// TwinCAT 3 PLC project pruebaFiltrado
// ProgramVersion: 3.1.4024.0
// libraries:
//   Tc2_Standard, * (Beckhoff Automation GmbH)
//   Tc2_System, * (Beckhoff Automation GmbH)
//   Tc3_Module, * (Beckhoff Automation GmbH)
// project tree:
//   GVLs/ GVLvars.TcGVL
//   / PlcTask.TcTTO
//   POUs/ MAIN.TcPOU
// real-time tasks:
//   TASK PlcTask: cycle T#10ms, priority 20, ADS port 350

CONFIGURATION pruebaFiltrado
    RESOURCE PLC ON TwinCAT3
        TASK PlcTask(INTERVAL := T#10ms, PRIORITY := 20);
        PROGRAM MAIN WITH PlcTask : MAIN;
    END_RESOURCE
END_CONFIGURATION

// ---- GVLs/GVLvars.TcGVL
{attribute 'qualified_only'}
VAR_GLOBAL
	// Cuadro
	{attribute 'OPC.UA.DA' := '1'}
	botonStart : BOOL;
	
	// Cintas
	{attribute 'OPC.UA.DA' := '1'}
	cintaVision : BOOL;
	{attribute 'OPC.UA.DA' := '1'}
	cintaRemoveVision : BOOL;
	{attribute 'OPC.UA.DA' := '1'}
	cintaBascula : BOOL;
	{attribute 'OPC.UA.DA' := '1'}
	cintaPostBascula : BOOL;
	{attribute 'OPC.UA.DA' := '1'}
	cintaRemoveBascula : BOOL;

	// Sensores
	{attribute 'OPC.UA.DA' := '1'}
	pesoBascula : REAL;
	{attribute 'OPC.UA.DA' := '1'}
 	sDifusoRemoveVision : BOOL;
	{attribute 'OPC.UA.DA' := '1'}
	sDifusoRemovePeso : BOOL;
	{attribute 'OPC.UA.DA' := '1'}
	sDifusoVision : BOOL;
 	{attribute 'OPC.UA.DA' := '1'}
	sDifusoBascula : BOOL;
	{attribute 'OPC.UA.DA' := '1'}
	sDifusoPostBascula : BOOL;
	{attribute 'OPC.UA.DA' := '1'}
 	sCilindroVision : BOOL;
	{attribute 'OPC.UA.DA' := '1'}
 	sCilindroBascula : BOOL;
	{attribute 'OPC.UA.DA' := '1'}
	sVision : INT;
	
	
	// Cilindros
	{attribute 'OPC.UA.DA' := '1'}
	sCilindroVisionDelantero : BOOL;
	{attribute 'OPC.UA.DA' := '1'}
	sCilindroVisionPosterior : BOOL;
	{attribute 'OPC.UA.DA' := '1'}
	sCilindroBasculaDelantero : BOOL;
	{attribute 'OPC.UA.DA' := '1'}
	sCilindroBasculaPosterior : BOOL;
	{attribute 'OPC.UA.DA' := '1'}
 	cilindroVision : BOOL;
	{attribute 'OPC.UA.DA' := '1'}
 	cilindroBascula : BOOL;
	
END_VAR

// ---- POUs/MAIN.TcPOU
PROGRAM MAIN
VAR
	enclaveStart: BOOL;
	cintaRemoveVision: BOOL;
	cintaBascula: BOOL;
	cintaPostBascula: BOOL;
	cintaRemoveBascula: BOOL;
	cintaVision: BOOL;
	timerVision: TON;
	
	descarteXcolor: BOOL;
	cilindroVision: BOOL;
	cintaDescarteVision: BOOL;
	timerBascula: TON;
	descarteXpeso: BOOL;
	cilindroBascula: BOOL;
	cintaDescarteBascula: BOOL;
END_VAR

(*

1 - Si se pulsa strart -> enclave y arranque de cintas

2 - Si se detecta en el sensor fotoelectrico de vision
	* Se para esa cinta 2 segundos
	* Se cogen las caracteristicas del objeto
		- Base azul : 3
		- Base verde : 6
		- Base metal : 9
	* En caso de descarte 
		- Se para cinta con el sensor delanterio del cilindro
		- Se acciona el cilindro
		- Se activa la cinta de descarte con el sensor fotoelectrico 
		  ( el tiempo de activo se sabe por vel y distancia x.ej)
 
3 - Si se detecta objeto en la cinta de pesaje (sensor fotoelectrico)
	* Se para la cinta 2 segundos
	* Se cogen als caracteristicas del objeto
		- Bases verde / azul : 7 kg
		- Base metalica : 9 kg
	* En caso de descarte
		--- Repetir proceso anterior

4 - Actualizar salidas

*)

// ------------------- PASO 1 -------------------

IF GVLvars.botonStart THEN
	enclaveStart := TRUE;
	cintaVision := TRUE;
	cintaRemoveVision := TRUE;
	cintaBascula := TRUE;
	cintaPostBascula := TRUE;
	cintaRemoveBascula 	:= TRUE;
END_IF


IF enclaveStart THEN
	
// ------------------- PASO 2 - Filtro Vision -------------------

	IF GVLvars.sDifusoVision THEN
		cintaVision := FALSE; // Se para la cinta
		timerVision(IN:=TRUE, PT:=T#2S);
			IF timerVision.Q THEN
				timerVision(IN:=FALSE);
				// Si es color azul o metalica continua 
				IF GVLvars.sVision = 3 OR GVLvars.sVision = 9 THEN
					descarteXcolor := FALSE;
				// Se descarta la base
				ELSE
					descarteXcolor := TRUE;
				END_IF
				cintaVision := TRUE; // Reanuda la marcha
				// Si hay que descratar y se detecta objeto delante del cilindro
				IF descarteXcolor AND GVLvars.sCilindroVision THEN
					cintaVision := FALSE;
					cilindroVision := TRUE;
					cintaDescarteVision := TRUE;
					// si e objeto ya esta en la cinta de descarte se reanuda con la de vision
					IF GVLvars.cintaRemoveVision THEN
						cintaVision := TRUE;
					END_IF
				END_IF
			END_IF
	END_IF
	
	
// ------------------ PASO 3 - Filtro peso -------------------

	IF GVLvars.sDifusoBascula THEN
		cintaBascula := FALSE; // Se para la cinta
		timerBascula(IN:=TRUE, PT:=T#2S);
			IF timerVision.Q THEN
				timerBascula(IN:=FALSE);
				// Si es color azul o metalica continua 
				IF GVLvars.pesoBascula > 8 THEN
					descarteXpeso := TRUE;
				// Se descarta la base
				ELSE
					descarteXpeso:= FALSE;
				END_IF
				cintaBascula := TRUE; // Reanuda la marcha
				// Si hay que descratar y se detecta objeto delante del cilindro
				IF descarteXpeso AND GVLvars.sCilindroBascula THEN
					cintaBascula := FALSE;
					cilindroBascula := TRUE;
					cintaDescarteBascula := TRUE;
					// si e objeto ya esta en la cinta de descarte se reanuda con la de vision
					// ANADIR LIMTES CILINDRO
					IF GVLvars.cintaRemoveBascula THEN
						cintaBascula := TRUE;
					END_IF
				END_IF
			END_IF
	END_IF

END_IF


// ----------------- PASO 4 ------------------

// Cintas
GVLvars.cintaBascula := cintaBascula;
GVLvars.cintaPostBascula := cintaPostBascula;
GVLvars.cintaRemoveBascula := cintaRemoveBascula;
GVLvars.cintaRemoveVision := cintaRemoveVision;
GVLvars.cintaVision := cintaVision;

// Cilindros
GVLvars.cilindroBascula := cilindroBascula;
GVLvars.cilindroVision := cilindroVision;

END_PROGRAM
